// TIA Portal project "2022.05.07-人机交互界面" (V17)

(* hardware
DEVICE "S7-1500/ET200MP station_1"  S7-1500 station
   slot 0: "导轨_0"  Rack  6ES7 590-1***0-0AA0
   slot 1: "PLC_1500"  CPU 1516-3 PN/DP  6ES7 516-3AN00-0AB0  V1.7
      slot 3: "CPU 显示_1"  6ES7591-1BA00-0AA0
      slot 32768: "PROFINET 接口_1"  X1
         slot 32769: "端口_1"  X1 P1
         slot 32770: "端口_2"  X1 P2
      slot 33024: "PROFINET 接口_2"  X2
         slot 33025: "端口_1"  X2 P1
      slot 33280: "DP 接口_1"  X3
   slot 2: "DI 32x24VDC BA_1"  DI 32x24VDC BA  6ES7 521-1BL10-0AA0  V1.1
   slot 3: "DQ 32x24VDC/0.5A HF_1"  DQ 32x24VDC/0.5A HF  6ES7 522-1BL01-0AB0  V1.1
DEVICE "HMI_1"  TP1200 Comfort
   slot 0: "HMI_1"  TP1200 Comfort  6AV2 124-0MC01-0AX0  17.0.0.0
   slot 1: "HMI_RT_1"  TP1200 Comfort  6AV2 124-0MC01-0AX0  17.0.0.0
   slot 5: "HMI_1.IE_CP_1"  PROFINET Interface  17.0.0.0
      slot 1: "PROFINET Interface_1"  PROFINET Interface
         slot 1: "Port_1"  Port
         slot 2: "Port_2"  Port
   slot 7: "HMI_1.MPI/DP_CP_1"  MPI/DP Interface  17.0.0.0
*)

// ===== PLC "PLC_1500"  CPU 1516-3 PN/DP =====

VAR_GLOBAL   // PLC tag table "默认变量表"
   "按钮1" AT %I0.0 : Bool;
   "按钮2" AT %I0.1 : Bool;
   "按钮3" AT %I0.2 : Bool;
   "按钮4" AT %I0.3 : Bool;
   "按钮5" AT %I0.4 : Bool;
   "按钮6" AT %I0.5 : Bool;
   "按钮7" AT %I0.6 : Bool;
   "按钮8" AT %I0.7 : Bool;
   "按钮9" AT %I1.0 : Bool;
   "按钮10" AT %I1.1 : Bool;
   "按钮11" AT %I1.2 : Bool;
   "指示灯1" AT %Q0.0 : Bool;
   "指示灯2" AT %Q0.1 : Bool;
   "指示灯3" AT %Q0.2 : Bool;
   "指示灯4" AT %Q0.3 : Bool;
   "指示灯5" AT %Q0.4 : Bool;
   "指示灯6" AT %Q0.5 : Bool;
   "指示灯7" AT %Q0.6 : Bool;
   "指示灯8" AT %Q0.7 : Bool;
   "指示灯9" AT %Q1.0 : Bool;
   "指示灯10" AT %Q1.1 : Bool;
   "指示灯11" AT %Q1.2 : Bool;
   "指示灯12" AT %Q1.3 : Bool;
END_VAR

ORGANIZATION_BLOCK "Main"   // OB1, LAD, ProgramCycle
TITLE = "Main Program Sweep (Cycle)"
{ S7_Optimized_Access := 'TRUE' }
VERSION : 0.1
   VAR_INPUT
      Initial_Call : Bool;   // Initial call of this OB
      Remanence : Bool;   // =True, if remanent data are available
   END_VAR
BEGIN

REGION Network 1: 1
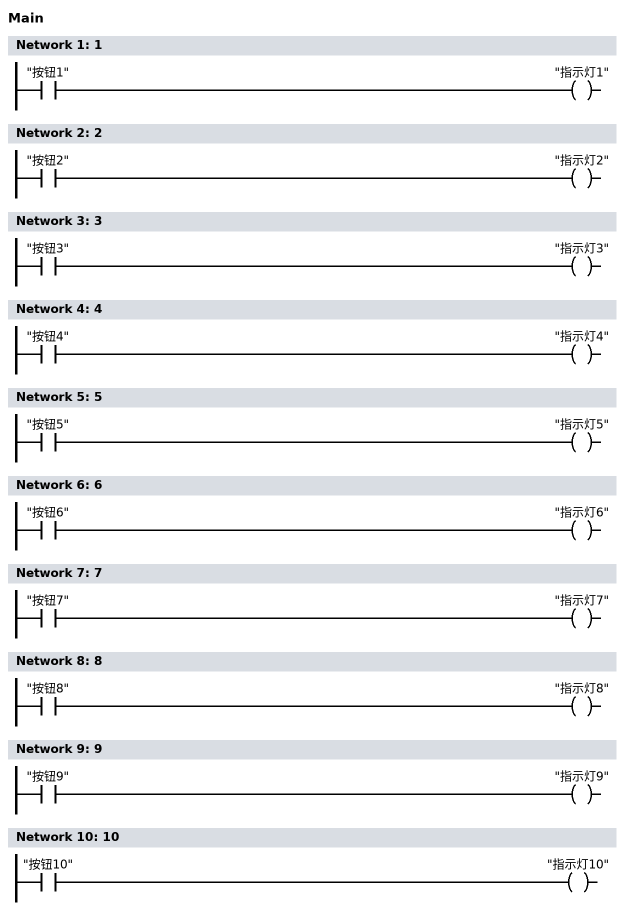
   RUNG wire#powerrail
      Contact( "按钮1" )
      Coil( "指示灯1" )
   END_RUNG
   // the same network as SCL:
   "指示灯1" := "按钮1";
END_REGION

REGION Network 2: 2
   RUNG wire#powerrail
      Contact( "按钮2" )
      Coil( "指示灯2" )
   END_RUNG
   // the same network as SCL:
   "指示灯2" := "按钮2";
END_REGION

REGION Network 3: 3
   RUNG wire#powerrail
      Contact( "按钮3" )
      Coil( "指示灯3" )
   END_RUNG
   // the same network as SCL:
   "指示灯3" := "按钮3";
END_REGION

REGION Network 4: 4
   RUNG wire#powerrail
      Contact( "按钮4" )
      Coil( "指示灯4" )
   END_RUNG
   // the same network as SCL:
   "指示灯4" := "按钮4";
END_REGION

REGION Network 5: 5
   RUNG wire#powerrail
      Contact( "按钮5" )
      Coil( "指示灯5" )
   END_RUNG
   // the same network as SCL:
   "指示灯5" := "按钮5";
END_REGION

REGION Network 6: 6
   RUNG wire#powerrail
      Contact( "按钮6" )
      Coil( "指示灯6" )
   END_RUNG
   // the same network as SCL:
   "指示灯6" := "按钮6";
END_REGION

REGION Network 7: 7
   RUNG wire#powerrail
      Contact( "按钮7" )
      Coil( "指示灯7" )
   END_RUNG
   // the same network as SCL:
   "指示灯7" := "按钮7";
END_REGION

REGION Network 8: 8
   RUNG wire#powerrail
      Contact( "按钮8" )
      Coil( "指示灯8" )
   END_RUNG
   // the same network as SCL:
   "指示灯8" := "按钮8";
END_REGION

REGION Network 9: 9
   RUNG wire#powerrail
      Contact( "按钮9" )
      Coil( "指示灯9" )
   END_RUNG
   // the same network as SCL:
   "指示灯9" := "按钮9";
END_REGION

REGION Network 10: 10
   RUNG wire#powerrail
      Contact( "按钮10" )
      Coil( "指示灯10" )
   END_RUNG
   // the same network as SCL:
   "指示灯10" := "按钮10";
END_REGION
END_ORGANIZATION_BLOCK

(* ===== HMI "HMI_RT_1" =====
system functions are stored by id; their names below are inferred from use
connection "PLC_1500": ETHERNET, S7_1500_OMS
connection "Connection_1": ETHERNET, S7_1500_OMS

HMI tags "默认变量表"
   "Tag_ScreenNumber" : UInt, internal

SlideinScreen "GraphX_Slidein_Left" 427x800
   TextField "文本域_1" at 70,190 size 83x29; Text '看法宝'

SlideinScreen "GraphX_Slidein_Bottom" 1280x267
   TextField "文本域_1" at 461,162 size 135x29; Text '你看不见我'

SlideinScreen "GraphX_Slidein_Right" 427x800
   TextField "文本域_1" at 231,379 size 83x29; Text '往这看'

SlideinScreen "GraphX_Slidein_Top" 1280x267
   TextField "文本域_1" at 349,62 size 109x29; Text '泰山压顶'

screen "根画面" 1280x740, template "模板_1"
   on GenerateScreen: SetTag("Tag_ScreenNumber", 1)
   TextField "HmiScreenItemData" at 78,282 size 1024x27; Text '欢迎进入 HMI_1 (TP1200 Comfort)！'

Template "模板_1" 1280x740
   Button "退出" at 1200,679 size 78x59; TextOff '退出'; PictureOff "ExitRuntime_TP1200_Comfort_TR"; PictureOn "ExitRuntime_TP1200_Comfort_TR"
      on Release: StopRuntime(0)
   Button "Template_Button" at 1120,679 size 78x59; TextOff 'Text'
   Button "Template_Button_1" at 1040,679 size 78x59; TextOff 'Text'
   Button "Template_Button_2" at 960,679 size 78x59; TextOff 'Text'
   Button "Template_Button_3" at 880,679 size 78x59; TextOff 'Text'
   Button "Template_Button_4" at 800,679 size 78x59; TextOff 'Text'
   Button "Template_Button_5" at 720,679 size 78x59; TextOff 'Text'
   Button "Template_Button_6" at 640,679 size 78x59; TextOff 'Text'
   Button "Template_Button_7" at 561,679 size 78x59; TextOff 'Text'
   Button "Template_Button_8" at 481,679 size 78x59; TextOff 'Text'
   Button "Template_Button_9" at 401,679 size 78x59; TextOff 'Text'
   Button "Template_Button_10" at 321,679 size 78x59; TextOff 'Text'
   Button "Template_Button_11" at 241,679 size 78x59; TextOff 'Text'
   Button "Template_Button_12" at 161,679 size 78x59; TextOff '第二个画面'
      on Click: ActivateScreen("画面_1", 0)
   Button "Template_Button_13" at 81,679 size 78x59; TextOff '第一个画面'
      on Click: ActivateScreen("根画面", 0)
   Button "起始画面" at 1,679 size 78x59; TextOff '起始画面'; PictureOff "NavigateHome_TP1200_Comfort_TR"; PictureOn "NavigateHome_TP1200_Comfort_TR"
      on Release: ActivateScreen("根画面", 0)
   Button "模板_按钮_1" at 426,50 size 148x50; TextOff '弹出画面'
      on Click: function_efd93a16("弹出画面_1", 100, 100, -1, -1, 1)
   Button "模板_按钮_2" at 426,124 size 148x50; TextOff '上侧滑入画面'
      on Click: function_cf6f4242("GraphX_Slidein_Top", -1)
   Button "模板_按钮_4" at 434,277 size 148x50; TextOff '下侧滑入画面'
      on Click: function_cf6f4242("GraphX_Slidein_Bottom", -1)
   Button "模板_按钮_5" at 239,186 size 148x50; TextOff '左侧滑入画面'
      on Click: function_cf6f4242("GraphX_Slidein_Left", -1)
   Button "模板_按钮_6" at 675,190 size 148x50; TextOff '右侧滑入画面'
      on Click: function_cf6f4242("GraphX_Slidein_Right", -1)

screen "画面_1" 1280x740
   TextField "文本域_1" at 218,80 size 125x27; Text '第二个画面'
*)